TYPE ST_PressureSensor :
STRUCT
	    nId             : INT;
    eZone           : E_ZoneId;
    rValueBar       : REAL;             // reading in bar
    rRateOfChange   : REAL;             // bar per minute
    eStatus         : E_SensorStatus;
    bAlarm          : BOOL;
    bHighHighAlarm  : BOOL;             // critical level
    bFault          : BOOL;
    bBypassed       : BOOL;
    tLastUpdate     : TIME;
    sLocation       : STRING;
END_STRUCT
END_TYPE

(* stored: Version 1.1.0.1, ProductVersion 3.1.4024.16
   DUT ST_PressureSensor: Id {42fff5ce-b4af-4445-928e-660c81cee5e5} *)
